// TIA Portal V19 export
DATA_BLOCK "Area0301_V_Counter"   // DB104
// stored: MemoryReserve 100
   VAR
      Value : LReal;
   END_VAR
BEGIN
END_DATA_BLOCK
